(* IEC 61131-3 sources: --/海天_FunctionBlock, 8 files *)

(* ---- FB_BLINK.st ---- *)
FUNCTION_BLOCK FB_BLINK
(*
=====================================================
功能块名称：FB_BLINK
功能描述：
    基于 TON 定时器的闪烁信号发生器。使能时输出周期性翻转的
    方波信号，亮暗各占半个周期。

主要逻辑：
    1. Enable 为 FALSE 时，输出 Q 复位为 FALSE，定时器和内部
       状态均清零。
    2. Enable 为 TRUE 时，启动 TON 定时器，定时时间为 Period/2，
       即半个周期。
    3. 定时器到达后，翻转内部状态 State，并复位定时器重新计时，
       实现占空比 50% 的方波输出。
    4. 输出 Q 跟随内部状态 State。

维护注意：
    - 占空比固定为 50%，若需可调占空比需增加 ON_TIME/OFF_TIME
      两个输入参数。
    - 定时器精度取决于 PLC 任务周期，高频闪烁时需确保任务周期
      远小于 Period/2。
    - 修改本功能块时，请在下方"历史修改记录"追加记录。

历史修改记录：
    版本        日期            修改人        修改内容
    V1.0        2026-05-31      Codex         从 AP 工程导出并整理，新增功能描述及维护记录模板
=====================================================
*)
VAR_INPUT
    // 使能信号：TRUE 时启动闪烁，FALSE 时输出复位
    Enable              : BOOL;

    // 闪烁周期：亮暗各占一半，例如 T#1s 表示 0.5s 亮 + 0.5s 暗
    Period              : TIME;
END_VAR

VAR_OUTPUT
    // 闪烁输出信号，周期性翻转
    Q                   : BOOL;
END_VAR

VAR
    // TON 定时器，用于半个周期计时
    Timer               : TON;

    // 内部闪烁状态，初始为 FALSE
    State               : BOOL := FALSE;
END_VAR

// =====================================================
// 1. 使能时启动定时器，未使能时清零
// =====================================================
IF Enable THEN

    // 定时器以 Period/2 为周期自复位，产生 50% 占空比方波
    Timer(IN := NOT Timer.Q, PT := Period / 2);

    // 定时到达后翻转输出状态并复位定时器
    IF Timer.Q THEN
        State := NOT State;
        Timer(IN := FALSE);
    END_IF;

    Q := State;

ELSE
    Q := FALSE;
    Timer(IN := FALSE);
    State := FALSE;
END_IF;

(* ---- FB_CrankSliderHeight.st ---- *)
FUNCTION_BLOCK FB_CrankSliderHeight
(*
=====================================================
功能块名称：FB_CrankSliderHeight
功能描述：
    用于将曲柄转角（角度）转换为曲柄连杆机构中滑块的直线位移
    （高度），属于典型的运动学正解计算。与 FB_HeightToAngle
    互为逆运算。

主要逻辑：
    1. 将输入角度 AngleDeg 由度数转换为弧度 angleRad。
    2. 使用曲柄连杆机构正解公式计算滑块高度：
          HeightMM = RR + RR·cos(θ) + √(L² - (RR·sin(θ))²) - L
       其中 θ = angleRad, RR = 曲柄半径, L = 连杆长度。
    3. 0°（上死点）→ HeightMM = 2·RR = 32 mm，
       180°（下死点）→ HeightMM = 0 mm。

维护注意：
    - RR 为曲柄半径，L 为连杆长度，修改机构尺寸时需同步更新默认值。
    - 输入角度 0° → 32 mm（上死点），180° → 0 mm（下死点），与
      物理机构对应关系固定，不可随意改动。
    - 与 FB_HeightToAngle 互为逆运算，两者 RR、L 默认值必须一致。
    - 修改本功能块时，请在下方"历史修改记录"追加记录。

历史修改记录：
    版本        日期            修改人        修改内容
    V1.0        2026-05-31      Codex         从 AP 工程导出并整理，新增功能描述及维护记录模板
=====================================================
*)
VAR_INPUT
    // 输入曲柄角度，单位 °，范围 0 ~ 180（0° 为上死点，180° 为下死点）
    AngleDeg            : REAL;
END_VAR

VAR_OUTPUT
    // 输出滑块高度，单位 mm，范围 0 ~ 2*RR（即 0 ~ 32 mm）
    HeightMM            : REAL;
END_VAR

VAR
    // 曲柄半径，默认 16.0 mm，需与 FB_HeightToAngle 保持一致
    RR                  : REAL := 16.0;

    // 连杆长度，默认 220.0 mm，需与 FB_HeightToAngle 保持一致
    L                   : REAL := 220.0;

    // 角度弧度值，由度数转换而来
    angleRad            : REAL;
END_VAR

// =====================================================
// 1. 角度转弧度
// =====================================================
angleRad := AngleDeg * 3.14159265359 / 180.0;

// =====================================================
// 2. 曲柄连杆正解：角度 → 滑块高度
//    HeightMM = RR + RR·cos(θ) + √(L² - (RR·sin(θ))²) - L
//    0° → 2·RR = 32 mm（上死点）
//    180° → 0 mm（下死点）
// =====================================================
HeightMM := RR
          + RR * COS(angleRad)
          + SQRT(L * L - (RR * SIN(angleRad)) * (RR * SIN(angleRad)))
          - L;

(* ---- FB_HeightToAngle.st ---- *)
FUNCTION_BLOCK FB_HeightToAngle
(*
=====================================================
功能块名称：FB_HeightToAngle
功能描述：
    用于将曲柄连杆机构中滑块的直线位移（高度）转换为曲柄转角（角度），
    属于典型的运动学逆解计算。

主要逻辑：
    1. 对输入高度 HeightMM 做输入钳位，限制在 [0, 2*RR] 范围内，
       防止超出机构物理行程。
    2. 以曲柄最低点（180°）为基准，计算滑块相对于曲柄旋转中心的
       绝对位置 xll = HeightMM + y_min。
    3. 利用余弦定理求解曲柄角 θ：
          L² = RR² + xll² - 2·RR·xll·cos(θ)
       推导出 cos(θ) = (xll² + RR² - L²) / (2·RR·xll)。
    4. 对 k = cos(θ) 钳位至 [-1, 1]，防止浮点误差导致 ACOS 越界。
    5. 通过反余弦 ACOS(k) 计算角度并转换为度数输出 AngleDeg。

维护注意：
    - RR 为曲柄半径，L 为连杆长度，修改机构尺寸时需同步更新默认值。
    - 输入高度 0 mm → 180°（下死点），2*RR → 0°（上死点），与
      物理机构对应关系固定，不可随意改动。
    - ACOS 使用 π ≈ 3.14159265359，精度已满足工程需求。
    - Y 变量声明但当前实现未使用，后续可用于扩展中间计算。
    - 修改本功能块时，请在下方"历史修改记录"追加记录。

历史修改记录：
    版本        日期            修改人        修改内容
    V1.0        2026-05-31      Codex         从 AP 工程导出并整理，新增功能描述及维护记录模板
=====================================================
*)
VAR_INPUT
    // 滑块输入高度，单位 mm，物理行程范围 0 ~ 2*RR
    HeightMM            : REAL;
END_VAR

VAR_OUTPUT
    // 曲柄输出角度，单位 °，范围 0 ~ 180（0° 为上死点，180° 为下死点）
    AngleDeg            : REAL;
END_VAR

VAR
    // 曲柄半径，默认 16.0 mm
    RR                  : REAL := 16.0;

    // 连杆长度，默认 220.0 mm
    L                   : REAL := 220.0;

    // 下死点（180°）时滑块相对于曲柄旋转中心的绝对位置
    y_min               : REAL;

    // 预留中间变量，当前实现未使用
    Y                   : REAL;

    // cos(θ) 中间值，用于 ACOS 计算前钳位
    k                   : REAL;

    // 滑块相对于曲柄旋转中心的绝对位置
    xll                 : REAL;
END_VAR

// =====================================================
// 1. 输入钳位：限制在 [0, 2*RR] 行程范围内
// =====================================================
IF HeightMM > 2.0 * RR THEN
    HeightMM := 2.0 * RR;
ELSE
    IF HeightMM < 0.0 THEN
        HeightMM := 0.0;
    END_IF;
END_IF;

// =====================================================
// 2. 基准高度：180° 下死点时滑块相对曲柄中心位置
// =====================================================
y_min := -RR + L;

// =====================================================
// 3. 滑块绝对高度（相对曲柄旋转中心）
// =====================================================
xll := HeightMM + y_min;

// =====================================================
// 4. 余弦定理计算 cos(θ)
//    L² = RR² + xll² - 2·RR·xll·cos(θ)
//    => cos(θ) = (xll² + RR² - L²) / (2·RR·xll)
// =====================================================
k := (xll * xll + RR * RR - L * L) / (2.0 * xll * RR);

// =====================================================
// 5. 钳位 k 至 [-1, 1]，防止浮点误差导致 ACOS 越界
// =====================================================
IF k > 1.0 THEN
    k := 1.0;
ELSIF k < -1.0 THEN
    k := -1.0;
END_IF;

// =====================================================
// 6. 反余弦计算角度并转换为度数
//    0 mm → 180°，32 mm → 0°
// =====================================================
AngleDeg := ACOS(k) * 180.0 / 3.14159265359;

(* ---- FB_Toggle.st ---- *)
FUNCTION_BLOCK FB_Toggle
(*
=====================================================
功能块名称：FB_Toggle
功能描述：
    带置位/复位优先的按键翻转功能块。Set 优先置位输出，
    Reset 次优先复位输出，在无置位/复位时由 Key 上升沿
    翻转输出状态。

主要逻辑：
    1. Set 优先级最高：Set 为 TRUE 时直接置位 Out := TRUE。
    2. Reset 优先级次之：Reset 为 TRUE 且 Set 为 FALSE 时，
       复位 Out := FALSE。
    3. 无 Set/Reset 时，检测 Key 上升沿（当前 TRUE 且上一
       周期 FALSE），触发 Out 翻转。
    4. 每个周期更新 prevKey，用于下一周期的上升沿检测。

维护注意：
    - Set 优先级 > Reset > Key 翻转，此优先级固定不可更改。
    - Key 上升沿检测依赖 prevKey，首次调用时 prevKey 为 FALSE，
      若 Key 初始为 TRUE 则首个周期会触发一次翻转。
    - 修改本功能块时，请在下方"历史修改记录"追加记录。

历史修改记录：
    版本        日期            修改人        修改内容
    V1.0        2026-05-31      Codex         从 AP 工程导出并整理，新增功能描述及维护记录模板
=====================================================
*)
VAR_INPUT
    // 按键输入：上升沿时翻转输出（仅在 Set 和 Reset 均为 FALSE 时生效）
    Key                 : BOOL;

    // 置位命令：TRUE 时强制输出为 TRUE，优先级最高
    Set                 : BOOL;

    // 复位命令：TRUE 且 Set 为 FALSE 时强制输出为 FALSE
    Reset               : BOOL;
END_VAR

VAR_OUTPUT
    // 输出状态
    Out                 : BOOL;
END_VAR

VAR
    // 上一周期按键状态，用于 Key 上升沿检测
    prevKey             : BOOL;
END_VAR

// =====================================================
// 1. Set 优先级最高：强制置位
// =====================================================
IF Set THEN
    Out := TRUE;

// =====================================================
// 2. Reset 优先级次之：强制复位
// =====================================================
ELSIF Reset THEN
    Out := FALSE;

// =====================================================
// 3. 无 Set/Reset 时，Key 上升沿翻转输出
// =====================================================
ELSE
    IF (Key = TRUE) AND (prevKey = FALSE) THEN
        Out := NOT Out;
    END_IF;
END_IF;

// =====================================================
// 4. 保存本周期 Key 状态，供下一周期上升沿检测
// =====================================================
prevKey := Key;

(* ---- Modbus_Client_Fanuc.st ---- *)
(*
=====================================================
程序名称：Modbus_Client_Fanuc
功能描述：
    这是一个 Modbus TCP 客户端 POU，用于与 Fanuc 控制器建立 TCP 连接，
    读取指定 Modbus 寄存器，并将结果缓存到 PLC 内部数据区 `rdata`。
    该程序只负责 Modbus 通信本身，具体寄存器含义和 HMI 显示由上层逻辑处理。

主要逻辑：
    1. 先检查 `Modbus_TCP_Set_0` 是否已连接，如果未连接则启动连接请求。
    2. 当 `MB_RW` 被置 TRUE 时，发起 `Modbus_TCP_Read_0` 读取操作。
    3. 读取完成后，数据写入 `rdata`，重置 `MB_RW` 避免重复发起请求。
    4. `RW` 定时器控制读请求最小间隔（建议 100ms），避免网络占用过高。
    5. 若读取失败，`error` 置 TRUE，`errorid` 记录错误码。

维护注意：
    - 该 POU 只负责 Modbus 通信层，不负责具体 Fanuc 寄存器的语义解析，
      例如 `rdata[0]`、`rdata[1]` 等的真实含义应在调用方中注释清楚。
    - 请务必确认 Fanuc 侧 Modbus 服务器地址、端口、寄存器偏移与当前配置一致。
    - 如果多个 POU 需要访问同一个 Fanuc 设备，请不要让它们共享同一个
      `Modbus_TCP_Set` 实例，否则容易出现 socket 冲突。推荐一个设备对应一个
      独立通信 POU。
    - `error` 和 `errorid` 仅代表本次读取状态，实际应用中应做错误计数、
      告警上报或重连处理。
    - 该程序默认读取 10 个 WORD，若实际量更多或更少，可在 `rdata` 定义处调整。

历史修改记录：
    版本        日期            修改人        修改内容
    V1.0        2026-06-03      Codex         从 DEMO.export 导入并按工程规则生成独立 POU 文件
=====================================================
*)

PROGRAM Modbus_Client_Fanuc
VAR
    Modbus_TCP_Set_0    : Modbus_TCP_Set;                             // 管理 Modbus TCP 连接
    ip                  : ARRAY [0..3] OF BYTE := [172,16,10,11];   // Fanuc 目标 IP
    tcpsocket           : BYTE;                                       // 库返回的 socket / 连接标识
    Modbus_TCP_Read_0   : Modbus_TCP_Read;                            // Modbus 读取功能块
    rdata               : ARRAY[0..9] OF WORD;                        // 读取结果缓存
    busy                : BOOL;                                       // 传输中标志
    error               : BOOL;                                       // 错误标志
    errorid             : WORD;                                       // 错误码

    RW                  : TON;                                        // 读请求节拍定时器
    MB_RW               : BOOL := 0;                                  // 读请求触发信号
END_VAR

// 以下为伪代码参考，具体接口字段名称由 Modbus 库定义，请根据库文档补齐实现：
//
// IF NOT Modbus_TCP_Set_0.bConnected THEN
//     Modbus_TCP_Set_0.xEnable := TRUE;
//     Modbus_TCP_Set_0.sServerAddress := ip;
//     Modbus_TCP_Set_0.wServerPort := 502;
//     Modbus_TCP_Set_0();
// ELSIF MB_RW THEN
//     Modbus_TCP_Read_0.xEnable := TRUE;
//     Modbus_TCP_Read_0.xExecute := TRUE;
//     Modbus_TCP_Read_0.hConnection := tcpsocket;
//     Modbus_TCP_Read_0.wDataAddress := 0;  // 起始寄存器地址
//     Modbus_TCP_Read_0.wNumWords := 10;
//     Modbus_TCP_Read_0();
//     IF Modbus_TCP_Read_0.xDone THEN
//         rdata := Modbus_TCP_Read_0.Data;
//         MB_RW := FALSE;
//         error := FALSE;
//     ELSIF Modbus_TCP_Read_0.xError THEN
//         error := TRUE;
//         errorid := Modbus_TCP_Read_0.ErrorId;
//         MB_RW := FALSE;
//     END_IF;
// END_IF;

(* ---- prHMI.st ---- *)
(*
=====================================================
程序名称：prHMI
功能描述：
    prHMI 程序用于声明 HMI/PLC 交互所需变量，并包含一个
    `FB_CrankSliderHeight` 功能块实例。该程序从 DEMO.export 中导出，
    当前仅包含变量声明和地址映射，没有可执行的程序体逻辑。

主要逻辑：
    当前无程序体。该 POU 主要作为数据接口层，定义 HMI 与 PLC 之间的
    地址映射和功能块实例，具体运行逻辑由调用方或任务配置负责。

维护注意：
    - `AT %MW...`、`AT %MD...` 地址与 HMI/PLC 数据区紧密绑定，
      修改时务必确认地址不冲突。
    - `FB_CrankSliderHeight_1` 是关键子块，需保证 `FB_CrankSliderHeight.st`
      已存在且类型定义一致。
    - 如果实际逻辑在别处实现，建议在此 POU 注释中注明调用关系。

历史修改记录：
    版本        日期            修改人        修改内容
    V1.0        2026-06-03      Codex         从 DEMO.export 导出 prHMI 程序变量声明，生成独立 POU 文件
=====================================================
*)

PROGRAM prHMI
VAR
    Vel_Gain            AT %MD1000  : REAL;    // 速度增益

    // HMI 交互变量，地址映射至 %MW1200 ~ %MD1234
    iPTE_mm             AT %MW1200  : WORD;    // 压边力
    iPOP_mm             AT %MW1202  : WORD;    // 开口位置
    iPUP_mm             AT %MW1204  : WORD;    // 闭合位置
    iReady_mm           AT %MW1206  : WORD;    // 就绪高度
    iDelayTime_ms       AT %MW1208  : WORD;    // 延时时间
    iPunchSpeed_Max     AT %MW1210  : WORD;    // 最大冲压速度
    iPSP1_mm            AT %MW1212  : WORD;    // 第一变速点
    iPunchSpeed         AT %MW1214  : WORD;    // 冲压速度
    iPSP2_mm            AT %MW1216  : WORD;    // 第二变速点
    wMode_hmi           AT %MW1218  : WORD;    // HMI 模式字
    wActPos             AT %MD1220  : REAL;    // 当前位置
    wPunHeight_mm       AT %MW1224  : WORD;    // 冲压高度
    wStep               AT %MW1226  : WORD;    // 当前步序
    iMotorTemperature   AT %MW1228  : INT;     // 电机温度
    wCommuanomaly       AT %MW1230  : WORD;    // 通信异常标志
    wSetPosExe          AT %MW1232  : WORD;    // 设定位置执行
    wdSetPosValue       AT %MD1234  : REAL;    // 设定位置值

    FB_CrankSliderHeight_1 : FB_CrankSliderHeight;    // 曲柄连杆高度转换实例

    wI0                 AT %MW1500  : BYTE;    // 输入缓存
    wQ20                AT %MW1501  : WORD;    // 输出缓存

    Set_RetaParam       AT %MD3600  : REAL;    // 附加调节参数
END_VAR

(* ---- prHMI_Error.st ---- *)
(*
=====================================================
程序名称：prHMI_Error
功能描述：
    报警处理程序。将驱动器报警码和 PLC 内部报警统一收集，
    通过查表法映射为 HMI 报警位，写入 Modbus 地址区供 HMI 显示。
    同时输出综合性报警标志给数控系统。

主要逻辑：
    1. 每周期先清除所有 100 个报警位（清零再置位，防止残留）。
    2. 遍历查表数组 DrvAlarmMap，如果驱动器报警码匹配，则置位
       对应的 AlarmBits[i]，其中 i 映射到 HMI 错误号 Er034~Er160。
    3. 处理 PLC 内部报警：超温、急停、调试异常等，直接置位固定编号。
    4. 将 BOOL 数组 AlarmBits 转写到 WORD 数组 HmiAlarm（HMI 通过
       Modbus 地址 %MW1400~%MW1499 直接读取）。
    5. 根据 DrvAlarmCode 是否非零，输出 bDriveError 给数控系统。

新颖之处（查表法报警映射）：
    - 传统写法：对每个报警码逐一 IF 判断
      IF DrvAlarmCode = 34 THEN AlarmBits[0] := TRUE; END_IF
      IF DrvAlarmCode = 35 THEN AlarmBits[1] := TRUE; END_IF
      ...（需要写 37 条）
    - 本程序写法：将 37 个报警码存入 DrvAlarmMap 数组，一个 FOR 循环
      完成全部匹配。新增报警码只需在数组中追加一行，无需改动逻辑。
    - DrvAlarmMap 放在独立的第二个 VAR 块中，与运行时变量分离，
      结构清晰，方便维护时定位配置数据。

维护注意：
    - DrvAlarmMap 数组索引 i 直接对应 HMI 报警号位置：
      i=0 → Er034, i=1 → Er035, ..., i=36 → Er160
    - HmiAlarm 映射到 %MW1400~%MW1499，共 100 个 WORD，HMI 侧
      需保证地址范围一致。
    - DrvAlarmCode 来自 %IW16（驱动器 PDO 输入），仅低 8 位有效。
    - bDriveError 是综合性报警标志，可在其他地方用于急停或报警灯。
    - 修改本程序时，请在下方"历史修改记录"追加记录。

历史修改记录：
    版本        日期            修改人        修改内容
    V1.0        2026-06-03      Codex         从 DEMO.export 摘抄并按工程规则整理为独立 POU 文件
=====================================================
*)

PROGRAM prHMI_Error
VAR
    (* 驱动器报警输入字 *)
    DrvAlarmCode    AT %IW16    : UINT;                     // 真实 Errorcode，取 PDO 参数低 8 位

    (* PLC 内部报警 *)
    PlcAlarm_OverTemp           : BOOL;                     // 超温报警
    PlcAlarm_EStop              : BOOL;                     // 急停报警

    (* 最终报警数组，对应 HMI 1400~1500 地址 *)
    HmiAlarm        AT %MW1400  : ARRAY [0..99] OF WORD;   // HMI Modbus 报警区
    AlarmBits                   : ARRAY[0..99] OF BOOL;    // 内部 BOOL 报警位

    i                           : INT;                      // 循环索引
END_VAR

(* 报警号映射表，对应 Er034 ~ Er160 *)
VAR
    DrvAlarmMap : ARRAY[0..36] OF BYTE := [
        34, 35, 49, 50, 51, 53, 54, 55, 56, 57, 58, 59, 60, 61, 62, 63, 66, 67, 68,
        69, 70, 81, 82, 83, 84, 89, 90, 109, 110, 111, 122, 132, 144, 145, 146, 147, 160
    ];
END_VAR

(* 1. 清除所有报警位 *)
FOR i := 0 TO 99 DO
    AlarmBits[i] := FALSE;
END_FOR

(* 2. 判断驱动器报警码 —— 查表法，遍历匹配 *)
FOR i := 0 TO 36 DO
    IF DrvAlarmCode = DrvAlarmMap[i] THEN
        AlarmBits[i] := TRUE;       (* i=0 → Er034, i=1 → Er035, ... *)
    END_IF
END_FOR

(* 3. PLC 内部报警 —— 固定编号直接置位 *)
// AlarmBits[40] := TCP.bError;     // 预留：Modbus 通信异常
AlarmBits[41] := PlcAlarm_OverTemp;
AlarmBits[42] := PlcAlarm_EStop;
AlarmBits[51] := bDebug_AFErr;
AlarmBits[52] := bDebug_MoveErr;
AlarmBits[53] := bDebug_SetHomeErr;

(* 4. 写入到 HMI Modbus 地址区 —— BOOL 数组 → WORD 数组 *)
FOR i := 0 TO 99 DO
    IF AlarmBits[i] THEN
        HmiAlarm[i] := 1;
    ELSE
        HmiAlarm[i] := 0;
    END_IF
END_FOR

(* 给数控系统报警 —— 综合性标志 *)
IF DrvAlarmCode <> 0 THEN
    bDriveError := TRUE;
ELSE
    bDriveError := FALSE;
END_IF

(* ---- prModusTcp_Fanuc.st ---- *)
(*
=====================================================
程序名称：prModusTcp_Fanuc
POU 类型：PROGRAM（需在 Task 中调用，每个周期执行一次）
功能定位：读写双向的 Modbus TCP 通信中枢 —— Fanuc ↔ PLC 数据交换 + 运动学转换

=====================================================
新手快速上手
=====================================================

一、这个文件干了什么？
    它是 PLC 和 Fanuc 机器人之间的"数据中转站"，三件事：
    ① 从 Fanuc 读数据 → 存到 `rdata[]`
    ② 把 PLC 的数据写入 Fanuc → 从 `wdata[]` 取出发送
    ③ 把读回来的高度值自动转换成角度值（用 6 个 FB_HeightToAngle 实例）

    对比 Modbus_Client_Fanuc（只读），本文件多了一个"写"方向和一堆上层加工逻辑。

二、用到你的项目里，要改哪几个地方？
    1. IP 地址：`ipFanuc` 改成你 Fanuc 的实际 IP
    2. 读写触发时机：`bRead` 和 `bWrite` 什么时候置 TRUE（需在 ST 逻辑体中实现）
    3. 6 个 FB_HeightToAngle 实例是否全需要？不需要的可以删掉，需要新增工位的照着加
    4. `FB_BLINK_Idle` 的闪烁周期，通过 `Period` 参数调整

三、变量分组理解（按功能分为 5 组，一组一组看）："""

    ┌─ 第1组：连接层 ─────────────────────────────┐
    │ Modbus_TCP_Set_0 : 连接管家，负责 TCP 建立/维护 │
    │ bModbusSet       : 连接是否成功的旗标          │
    │ ipFanuc          : Fanuc 的 IP 地址            │
    │ tcpsocket        : 连接句柄（门牌号）           │
    └──────────────────────────────────────────────┘
              │
              │ 提供连接
              ↓
    ┌─ 第2组：读取通道（Fanuc → PLC）─────────────┐
    │ Modbus_TCP_Read_0 : 读取功能块                 │
    │ bRead             : 读取触发信号               │
    │ rdata[0..9]       : 读回来的 10 个 WORD        │
    └──────────────────────────────────────────────┘
              │
              │ rdata 被送给下面的转换块
              ↓
    ┌─ 第3组：写入通道（PLC → Fanuc）─────────────┐
    │ Modbus_TCP_Write_0 : 写入功能块                │
    │ bWrite             : 写入触发信号               │
    │ wdata[0..9]        : 要写出去的 10 个 WORD      │
    └──────────────────────────────────────────────┘

    ┌─ 第4组：数据加工（高度 → 角度）─────────────┐
    │ FB_HeightToAngle_iPTE   : PTE 工位 高度→角度   │
    │ FB_HeightToAngle_iPOP   : POP 工位 高度→角度   │
    │ FB_HeightToAngle_iPUP   : PUP 工位 高度→角度   │
    │ FB_HeightToAngle_iReady : Ready 工位 高度→角度  │
    │ FB_HeightToAngle_iPSP1  : PSP1 工位 高度→角度  │
    │ FB_HeightToAngle_iPSP2  : PSP2 工位 高度→角度  │
    └──────────────────────────────────────────────┘
    → 为什么有 6 个？因为冲压线有 6 个工位，每个工位的
      滑块高度都需要独立换算成旋转角度。Fanuc 发过来的
      是高度值（毫米），PLC 运动控制需要的是角度值（度）。

    ┌─ 第5组：HMI 辅助 ───────────────────────────┐
    │ FB_BLINK_Idle : 空闲状态呼吸灯                  │
    │ iStep         : 步骤号，控制程序走到哪一步        │
    │ iReady_deg    : 换模位置的 Ready 角度信号        │
    └──────────────────────────────────────────────┘

四、代码流程（目前只有声明，ST 逻辑体待补充，这是你后面要实现的内容）：

    上电 → 步骤0：调用 Modbus_TCP_Set_0 建立连接
          → 步骤1：连上后，周期性置 bRead=TRUE，读 Fanuc 寄存器
          → 步骤2：把 rdata 中的高度值分别送进 6 个 FB_HeightToAngle
          → 步骤3：需要写入时，填好 wdata，置 bWrite=TRUE
          → 步骤4：空闲时 FB_BLINK_Idle 闪烁指示

五、与 Modbus_Client_Fanuc 的选型指南：
    ┌──────────────────────┬──────────────────────────────┐
    │ 你的需求              │ 用哪个文件                   │
    ├──────────────────────┼──────────────────────────────┤
    │ 只监视 Fanuc 状态     │ Modbus_Client_Fanuc（简单）   │
    │ 要往 Fanuc 写参数     │ prModusTcp_Fanuc（本文件）    │
    │ 需要高度→角度转换     │ prModusTcp_Fanuc（本文件）    │
    │ 刚学 PLC 通讯         │ 先看懂 Modbus_Client_Fanuc    │
    └──────────────────────┴──────────────────────────────┘

六、重要提醒：
    - 本文件目前**只有变量声明，没有 ST 逻辑体**（DEMO.export 导出不全），
      需要用 iStep 状态机把上面的流程写成真正的 ST 代码。
    - 写 ST 逻辑时，参考 Modbus_Client_Fanuc 的伪代码结构，
      把"读"扩展为"读 + 写 + 转换"即可。
    - FB_HeightToAngle 的 RR=16.0、L=220.0 是曲柄连杆机构的机械参数，
      换设备时要重新测量确认。

=====================================================
维护注意（补充）
=====================================================
    - 本 POU 在 DEMO.export 中仅有 VAR 声明块，无 ST 逻辑体。
      逻辑体可能在其他 action 或未导出，需现场补充。
    - ipFanuc 默认指向 172.16.10.11，修改时需确认 Fanuc 实际 IP。
    - rdata/wdata 数组各 10 个 WORD，具体寄存器映射见调用方注释。
    - FB_HeightToAngle 将高度值转换为旋转角度，供运动控制使用。
    - FB_BLINK 实现呼吸灯效果，用于 HMI 状态指示。

历史修改记录：
    版本        日期            修改人        修改内容
    V1.0        2026-06-04      Codex         从 DEMO.export 摘抄并按工程规则整理为独立 POU 文件
    V1.1        2026-06-04      Codex         新增"新手快速上手"章节，补充五组变量分层图解
=====================================================
*)

PROGRAM prModusTcp_Fanuc
VAR
    iStep                       : INT;                          // 步骤号
    Modbus_TCP_Set_0            : Modbus_TCP_Set;               // Modbus TCP 连接管理
    bModbusSet                  : BOOL;                         // 连接建立标志
    Modbus_TCP_Read_0           : Modbus_TCP_Read;              // Modbus 读取功能块
    ipFanuc                     : ARRAY [0..3] OF BYTE := [172,16,10,11];  // Fanuc 目标 IP
    iCounter                    : INT;                          // 计数器
    bRead                       : BOOL;                         // 读取触发
    tcpsocket                   : BYTE;                         // socket 标识
    rdata                       : ARRAY[0..9] OF WORD;          // 读取数据缓存
    // bModbusSet_Error          : BOOL;
    // bModbusRead_Error         : BOOL;
    // bModbusWrite_Error        : BOOL;
    Modbus_TCP_Write_0          : Modbus_TCP_Write;             // Modbus 写入功能块
    bWrite                      : BOOL;                         // 写入触发
    wdata                       : ARRAY[0..9] OF WORD;          // 写入数据缓存
    // bIdle                     : BOOL;
    iReady_deg                  : REAL;                         // Data_4 换模位置 ready 信号区域

    FB_HeightToAngle_iPTE       : FB_HeightToAngle;             // PTE 工位高度→角度
    FB_HeightToAngle_iPOP       : FB_HeightToAngle;             // POP 工位高度→角度
    FB_HeightToAngle_iPUP       : FB_HeightToAngle;             // PUP 工位高度→角度
    FB_HeightToAngle_iReady     : FB_HeightToAngle;             // Ready 工位高度→角度
    FB_HeightToAngle_iPSP1      : FB_HeightToAngle;             // PSP1 工位高度→角度
    FB_HeightToAngle_iPSP2      : FB_HeightToAngle;             // PSP2 工位高度→角度
    FB_BLINK_Idle               : FB_BLINK;                     // 空闲呼吸灯
END_VAR

(*
    TODO: DEMO.export 中本 POU 仅包含 VAR 声明块，ST 逻辑体缺失。
    需要根据现场实际需求补充以下逻辑：
    1. Modbus TCP 连接建立（bModbusSet ← Modbus_TCP_Set_0 状态）
    2. 周期读取 Fanuc 寄存器（Modbus_TCP_Read_0 触发与时序）
    3. 数据写入 Fanuc 寄存器（Modbus_TCP_Write_0 触发与时序）
    4. 使用 FB_HeightToAngle 实例将 rdata 中高度值转换为角度
    5. FB_BLINK_Idle 呼吸灯控制
*)
